// ---- FBs/Zaptec ECS/Client FBs/FB_ECS_HTTP_ZaptecAccount.TcPOU
{attribute 'hide_all_locals'}
FUNCTION_BLOCK FB_ECS_HTTP_ZaptecAccount
VAR_INPUT
	bStart					: BOOL;													//Start/Stop this Functions
	byMode					: BYTE;													//Work mode : 0 = Send current to each Charger; 1 = Send current to a Installation of chargers
	sUsername				: STRING(100);											//Username from the Zaptec Account
	sPassword				: STRING(100);											//Password from the Zaptec Account
	arrCharger				: ARRAY[1..100] OF ST_Zaptec_Input_Charger;				//Structure with Data for each Charging Station
	arrInstallation			: ARRAY[1..100] OF ST_Zaptec_Input_Installation;		//Structure with Data for each Installation of Charging Stations
END_VAR
VAR_OUTPUT
	bValidResult			: BOOL;													//Valid Result received from Server
	bBusy             		: BOOL;													//Busy Flag
    bError              	: BOOL;													//Error Flag
	hrErrorCode       		: HRESULT;												//Error Result from Http Client
	arrStateCharger			: ARRAY[1..100] OF ST_Zaptec_ECS_State;					//Output Structure with the State from each Charging Station
END_VAR
VAR
	fbHttpClient        	: FB_IotHttpClient :=(sHostName:='api.zaptec.com',		//Http Client Function
                       		  bKeepAlive:=FALSE, tConnectionTimeout:=T#10S);
	fbHttpPostToken         : FB_HTTP_Post_Zaptec_ReqToken;							//Http Post to receive the Bearer Token
 	fbHttpGetChrgState		: FB_HTTP_Get_Zaptec_ECS_State;							//Http Get to receive the State from each Charging station
	fbHttpPostCurrent		: FB_HTTP_Post_Zaptec_Current;							//Http Post to control each Chrging station or a installation of charging stations with the current setpoint
	fbTaskIndex				: GETCURTASKINDEX;										//Function to find the Task Index
	timDelay				: TON;													//Timer for Delay between the Requests
	timTimout				: TON;													//Timer for Timeout in the State machine
	timToken				: TON;													//Timer to make a Request for a new Token
	FPStart					: R_TRIG;												//Internal positive Edge
	FPErrorToken			: R_TRIG;												//Internal positive Edge
	FPErrorGetState			: R_TRIG;												//Internal positive Edge
	FPErrorPostCurrent		: R_TRIG;												//Internal positive Edge
	FPErrorClient			: R_TRIG;												//Internal positive Edge
	FPTimToken				: R_TRIG;												//Internal positive Edge
	FNStart					: F_TRIG;												//Internal negative Edge
	byNumberOfChargers		: BYTE;													//Number of charging station with insert ID in the Input Array
	byNumberOfInstallation	: BYTE;													//Number of Installations with insert ID in the Input Array
	byECSInProgress			: BYTE;													//Charging station in Progress to read out the State or write the current
	byInstInProgress		: BYTE;													//Installation of charging stations in Progress to write the current
	byLPInfo				: BYTE;													//Loop Variable to define some parts in the Code
	iState					: INT;													//Variabel for state machine
	iState_CP				: INT;													//Variabel for state machine to compare it for timeout
	udiCycleTime			: UDINT;												//Cycletime in ms
END_VAR

//Creator : Kai Ebensperger
//Company : Lynus AG
//Date : 04.11.2021
//Version : 1.0.0.0

//With this Function its possible to receive information from each charging station in a Zaptec Account in there cloudplattform
//Its also possible to control the charging station with this function by a curretn setpoint.
//We can control each Cahrging station with the current or each installation with more charging stations with a sum of current
//When the Installation mode is active, then the system of the charging station distribute the sum of current among themselves
//Attention : This Function need allways the Charging IDs. Even if the current is sent to the installation. Becasue the State Get Request for each charging station its possible only with the Charging IDs
//This Function can handle maximal 100 charging stations and 100 Installations

(*------------------------------------------------------------------------------------Limits------------------------------------------------------------------------------------------------------*)

byMode := LIMIT(0,byMode,1);

(*------------------------------------------------------------------------------------Configure HTTP Client------------------------------------------------------------------------------------------------------*)

IF NOT fbHttpClient.bConfigured THEN
    fbHttpClient.nHostPort:= 443;
	fbHttpClient.stTLS.bNoServerCertCheck := TRUE;
END_IF

(*------------------------------------------------------------------------------------Logic------------------------------------------------------------------------------------------------------*)

//Calculate the number of chargers and installations from the input array
byNumberOfChargers := 0;
	byNumberOfInstallation := 0;

FOR byLPInfo := 1 TO 100 BY 1 DO
	IF arrCharger[byLPInfo].sChargerID <> '' THEN byNumberOfChargers := byNumberOfChargers + 1; END_IF 
		IF arrInstallation[byLPInfo].sInstallationID <> '' THEN byNumberOfInstallation := byNumberOfInstallation + 1; END_IF  
END_FOR 	

//Delay between the Requests
fbTaskIndex(index=> );
	udiCycleTime := TwinCAT_SystemInfoVarList._TaskInfo[fbTaskIndex.index].CycleTime / 10000;
		timDelay(IN:= , PT:= T#1MS * udiCycleTime, Q=> , ET=> );

//Timout
IF iState_CP = iState AND iState <> 0 THEN timTimout.IN := TRUE; ELSE timTimout.IN := FALSE; END_IF
	timTimout(IN:= , PT:= T#20S, Q=> , ET=> );

//Timer for the Token
//After received the validation from the Token start this timer.
//After the Delay stop the State machine and make a request for a new Token
IF fbHttpPostToken.udiValidityToken <> 0 THEN
	timToken.PT := (T#1S * (fbHttpPostToken.udiValidityToken - 600));	//Less 10 Minutes
ELSE
	timToken.PT := T#600S;
END_IF
	timToken(IN:= , PT:= , Q=> , ET=> );	

FPTimToken(CLK:= timToken.Q, Q=> );
	
//Start	
FPStart(CLK:= bStart, Q=> );
	IF FPStart.Q AND NOT fbHttpPostToken.bBusy AND NOT fbHttpGetChrgState.bBusy AND NOT fbHttpPostCurrent.bBusy AND fbHttpClient.bConfigured THEN istate := 1; END_IF
		IF NOT bStart THEN istate := 0; END_IF	

CASE iState OF

	0://Init Step	
		fbHttpPostToken.bPostToken := FALSE;
			fbHttpGetChrgState.bSend := FALSE;
				fbHttpPostCurrent.bSend := FALSE;	
					byECSInProgress := 0;
						byInstInProgress := 0;
							timToken.IN := FALSE;
								bValidResult := FALSE;
									timdelay.IN := FALSE;
		
		FOR byLPInfo := 1 TO 100 BY 1 DO					
			arrStateCharger[byLPInfo].bIsEnabled := FALSE;	
				arrStateCharger[byLPInfo].bIsOnline := FALSE;
					arrStateCharger[byLPInfo].diOperationMode := 0;	
						arrStateCharger[byLPInfo].diWarnings := 0;
							arrStateCharger[byLPInfo].rAllocatedCurrent := 0;
								arrStateCharger[byLPInfo].rMaxCurrect := 0;
									arrStateCharger[byLPInfo].rMinCurrect := 0;
										arrStateCharger[byLPInfo].rCurrentL1 := 0;	
											arrStateCharger[byLPInfo].rCurrentL2 := 0;	
												arrStateCharger[byLPInfo].rCurrentL3 := 0;	
													arrStateCharger[byLPInfo].rPower := 0;
														arrStateCharger[byLPInfo].rEnergySession := 0;		
															arrStateCharger[byLPInfo].sChargerID := '';	
		END_FOR		
				
	1://Request for Bearer Token
		iState_CP := iState;
	
		fbHttpPostToken.bPostToken := TRUE;
			timToken.IN := FALSE;
		
		IF NOT fbHttpPostToken.bBusy THEN timdelay.IN := TRUE; END_IF 
	
		IF NOT fbHttpPostToken.bBusy AND fbHttpPostToken.bValidResult AND NOT fbHttpPostToken.bError AND timdelay.Q THEN
			istate := 2; 
				timdelay.IN := FALSE;
					byECSInProgress := 1;
						byInstInProgress := 1;
							fbHttpPostToken.bPostToken := FALSE;
								timToken.IN := TRUE;
		END_IF
		
		//Valid Result
		bValidResult := fbHttpPostToken.bValidResult;
		
		//Error, Timout or Request for a new Token
		IF FPErrorToken.Q OR timTimout.Q OR FPTimToken.Q OR FPErrorClient.Q THEN istate := 300; END_IF

	2://Request for State of Each Charging Station
		iState_CP := iState;
		
		fbHttpGetChrgState.bSend := TRUE;
			fbHttpGetChrgState.sChargerID := arrCharger[byECSInProgress].sChargerID;
		
		IF NOT fbHttpGetChrgState.bBusy THEN timdelay.IN := TRUE; END_IF 
		
		IF NOT fbHttpGetChrgState.bBusy AND fbHttpGetChrgState.bValidResult AND NOT fbHttpGetChrgState.bError AND timdelay.Q THEN
			IF byMode = 0 THEN istate := 3; END_IF
				IF byMode = 1 THEN istate := 4; END_IF
					timdelay.IN := FALSE;
						arrStateCharger[byECSInProgress] := fbHttpGetChrgState.stChargerStates;
							fbHttpGetChrgState.bSend := FALSE;	
		END_IF
		
		//Valid Result
		bValidResult := fbHttpGetChrgState.bValidResult;
		
		//Error, Timout or Request for a new Token
		IF FPErrorGetState.Q OR timTimout.Q OR FPTimToken.Q OR FPErrorClient.Q THEN istate := 300; END_IF
		
	3://Write current to charging station
		iState_CP := iState;
		
		fbHttpPostCurrent.bSend := TRUE;
			fbHttpPostCurrent.sID := arrCharger[byECSInProgress].sChargerID;
				fbHttpPostCurrent.rMaxCurrentCharger := arrCharger[byECSInProgress].rMaxCurrentCharger;
 					fbHttpPostCurrent.rMinCurrentCharger := arrCharger[byECSInProgress].rMinCurrentCharger;
		
		IF NOT fbHttpPostCurrent.bBusy THEN timdelay.IN := TRUE; END_IF 
		
		IF NOT fbHttpPostCurrent.bBusy AND fbHttpPostCurrent.bValidResult AND NOT fbHttpPostCurrent.bError AND timdelay.Q THEN
			iState := 5;
				timdelay.IN := FALSE;
					fbHttpPostCurrent.bSend := FALSE;	
		END_IF
		
		//Valid Result
		bValidResult := fbHttpPostCurrent.bValidResult;
		
		//Error, Timout or Request for a new Token
		IF FPErrorPostCurrent.Q OR timTimout.Q OR FPTimToken.Q OR FPErrorClient.Q THEN istate := 300; END_IF
		
	4://Write current to installation of charging stations	
		iState_CP := iState;	
	
		fbHttpPostCurrent.bSend := TRUE;
			fbHttpPostCurrent.sID := arrInstallation[byInstInProgress].sInstallationID;
				fbHttpPostCurrent.rAvailableCurrentInstallation := arrInstallation[byInstInProgress].rAvailableCurrentInstallation;
		
		IF NOT fbHttpPostCurrent.bBusy THEN timdelay.IN := TRUE; END_IF 
		
		IF NOT fbHttpPostCurrent.bBusy AND fbHttpPostCurrent.bValidResult AND NOT fbHttpPostCurrent.bError AND timdelay.Q THEN
			iState := 5;
				timdelay.IN := FALSE;
					fbHttpPostCurrent.bSend := FALSE;	
		END_IF
		
		//Valid Result
		bValidResult := fbHttpPostCurrent.bValidResult;
		
		//Error, Timout or Request for a new Token
		IF FPErrorPostCurrent.Q OR timTimout.Q OR FPTimToken.Q OR FPErrorClient.Q THEN istate := 300; END_IF
		
	5://Next charging station and next installation	
		iState_CP := iState;
		
		byECSInProgress := byECSInProgress + 1;
		byInstInProgress := byInstInProgress + 1;
		
		//Back to read out next state from charging station
		iState := 2;
		
		IF byECSInProgress > byNumberOfChargers THEN byECSInProgress := 1; END_IF
			IF byInstInProgress > byNumberOfInstallation THEN byInstInProgress := 1; END_IF  	
		
		//Reset Error
		bError := FALSE;
			
	300://Error or restart after receive a new Token
		iState_CP := iState;
		
		timdelay.IN := FALSE;
			fbHttpPostToken.bPostToken := FALSE;
				fbHttpGetChrgState.bSend := FALSE;
					fbHttpPostCurrent.bSend := FALSE;	
						byECSInProgress := 0;
							byInstInProgress := 0;
								bError := TRUE;
								//Restart
								IF NOT fbHttpPostToken.bBusy AND NOT fbHttpGetChrgState.bBusy AND NOT fbHttpPostCurrent.bBusy THEN 
									istate := 1;
								END_IF	
		
		
END_CASE		
		
(*------------------------------------------------------------------------------------HTTP Functions------------------------------------------------------------------------------------------------------*)

fbHttpPostToken(
	sUsername:= sUsername, 
	sPassword:= sPassword, 
	bPostToken:= , 
	tTimeOut:= T#20S,
	fbClient:= fbHttpClient, 
	bValidResult=> , 
	bBusy=> , 
	bError=> , 
	udiValidityToken=> , 
	sToken=> , 
	sTokenType=> );

FPErrorToken(CLK:= fbHttpPostToken.bError, Q=> );
	
fbHttpGetChrgState(
	bSend:= , 
	sToken:= fbHttpPostToken.sToken, 
	sTokenType:= fbHttpPostToken.sTokenType, 
	sChargerID:= , 
	tTimeOut:= T#20S,
	fbClient:= fbHttpClient, 
	bValidResult=> , 
	bBusy=> , 
	bError=> , 
	stChargerStates=> );

FPErrorGetState(CLK:= fbHttpGetChrgState.bError, Q=> );
	
fbHttpPostCurrent(
	bSend:= , 
	byMode:= byMode, 
	rMaxCurrentCharger:= , 
	rMinCurrentCharger:= , 
	rAvailableCurrentInstallation:= , 
	sToken:= fbHttpPostToken.sToken, 
	sTokenType:= fbHttpPostToken.sTokenType, 
	sID:= , 
	tTimeOut:= T#20S,
	fbClient:= fbHttpClient, 
	bValidResult=> , 
	bBusy=> , 
	bError=> );

FPErrorPostCurrent(CLK:= fbHttpPostCurrent.bError, Q=> );	

//Http Client
FNStart(CLK:= bStart, Q=> );
	IF FNStart.Q THEN fbHttpClient.Disconnect(); END_IF

fbHttpClient.Execute();

FPErrorClient(CLK:= fbHttpClient.bError, Q=> );

//Busy
IF fbHttpPostToken.bBusy OR fbHttpGetChrgState.bBusy OR fbHttpPostCurrent.bBusy THEN bBusy := TRUE; ELSE bBusy := FALSE; END_IF  

//Error
hrErrorCode := fbHttpClient.hrErrorCode;

END_FUNCTION_BLOCK

// ---- FBs/Zaptec ECS/Helper FBs/FB_HTTP_Post_Zaptec_ReqToken.TcPOU
{attribute 'hide_all_locals'}
{attribute 'conditionalshow'}
FUNCTION_BLOCK FB_HTTP_Post_Zaptec_ReqToken
VAR_INPUT
	{attribute 'hide'}
	sUsername			: STRING(100);											//Username from the Zaptec Account
	{attribute 'hide'}
	sPassword			: STRING(100);											//Password from the Zaptec Account
	{attribute 'hide'}
    bPostToken          : BOOL;													//Send Post Request for Token		
	{attribute 'hide'}
	tTimeOut			: TIME := T#10S;										//Timer for Timeout
END_VAR
VAR_IN_OUT
	{attribute 'hide'}
    fbClient            : FB_IotHttpClient;										//FB Http Client
END_VAR
VAR_OUTPUT
	{attribute 'hide'}
	bValidResult		: BOOL;													//Valid Result received from Server
	{attribute 'hide'}
	bBusy             	: BOOL;													//Busy Flag
	{attribute 'hide'}
    bError              : BOOL;													//Error Flag
	{attribute 'hide'}
	udiValidityToken	: UDINT;												//Validity from the Token in seconds. (Token is valid only for this time)
	{attribute 'hide'}
	sToken				: STRING(1500);											//Bearer Token
	{attribute 'hide'}
	sTokenType			: STRING(50);											//Token Type
END_VAR
VAR
	fbJsonRead			: FB_JsonDomParser;										//Json Parser
	jsonDoc		  		: SJsonValue;											//Json Value
	jsonProp			: SJsonValue;											//Json Value
    fbRequest           : FB_IotHttpRequest;									//HTTP Request
	fbHeader            : FB_IotHttpHeaderFieldMap;								//Header Function
	timTimeout			: TON;													//Timer for Timeout
    RisingEdge          : R_TRIG;												//Internal Risig Edge
    bOnce               : BOOL:= TRUE;											//Add the addidional Header Part
    bGetContentResult   : BOOL;													//Content Received
 	nState              : UDINT;												//State
	nReqCount           : UDINT;												//Request Counter
    nResCount           : UDINT;												//Receive Conter
    nValidResCount      : UDINT;												//Valid receive Counter
    nErrCount           : UDINT;												//Error Counter
	sUsernameInt		: STRING(200);											//Internal Username
	sPasswordInt		: STRING(200);											//Internal Password
   	sContent            : STRING(500);											//Content to send with the psot request
	sReceiveContent		: STRING(2000);											//Received Content
END_VAR

//Creator : Kai Ebensperger
//Company : Lynus AG
//Date : 03.11.2021
//Version : 1.0.0.0

//With this Function is possible to make a POST Request to a Zaptec Account to receive the Bearer Token
//This Token is neccessary for all other Requests to the Zaptec Account
//Each Token has a Validity

RisingEdge(CLK:= bPostToken);

//Content with Username and PW
sUsernameInt := sUsername;
sPasswordInt := sPassword;

//URL Encoding for Username
IF FIND(sUsernameInt,'@') <> 0 THEN
	sUsernameInt := REPLACE(sUsernameInt,'%40',1,FIND(sUsernameInt,'@'));
END_IF

//URL Encoding for Password
IF FIND(sPasswordInt,'@') <> 0 THEN
	sPasswordInt := REPLACE(sPasswordInt,'%40',1,FIND(sPasswordInt,'@'));
END_IF

//Prepear the Payload for the Post Request to receive the Token
sContent := 'grant_type=password&username=';
	CONCAT2(ADR(sContent),ADR(sUsernameInt),ADR(sContent),SIZEOF(sContent));
		sContent := CONCAT(sContent,'&password=');
			CONCAT2(ADR(sContent),ADR(sPasswordInt),ADR(sContent),SIZEOF(sContent));

//Add the Content type in the Header
IF bOnce THEN
    fbHeader.AddField('content-type','application/x-www-form-urlencoded', FALSE);
    bOnce:= FALSE;
END_IF

//Timer for Timeout
timTimeout(IN:= nState = 1 AND bBusy, PT:= tTimeOut, Q=> , ET=> );
	IF timTimeout.Q THEN nState := 0; bBusy := FALSE; END_IF

CASE nState OF
	
	0://Request
		IF RisingEdge.Q THEN
			IF fbRequest.SendRequest(sUri:= '/oauth/token', fbClient:= fbClient, 
									 eRequestType:= ETcIotHttpRequestType.HTTP_POST, 
									 pContent:= ADR(sContent), 
									 nContentSize:= LEN2(ADR(sContent)), fbHeader) THEN
				nState:= 1;
				nReqCount:= nReqCount+1;
				bBusy:= TRUE;
				bError:= FALSE;
				bValidResult := FALSE;
			END_IF
		END_IF
		
	1://Wait for the Response
		IF NOT fbRequest.bBusy THEN
			bError:= TRUE;
			IF NOT fbRequest.bError THEN
				bGetContentResult:= fbRequest.GetContent(pContent:= ADR(sReceiveContent),
														 nContentSize:= SIZEOF(sReceiveContent), 
														 bSetNullTermination:= TRUE);
				IF fbRequest.nStatusCode >= 200 AND fbRequest.nStatusCode < 300 THEN
					bValidResult := TRUE;
					//Parse Document
					jsonDoc := fbJsonRead.ParseDocument(sReceiveContent);
						//Token
						jsonProp := fbJsonRead.FindMember(jsonDoc,'access_token');
							IF jsonProp <> 0 AND fbJsonRead.IsString(jsonProp) THEN
								fbJsonRead.CopyString(jsonProp,sToken,SIZEOF(sToken));	
							END_IF
						//Token Type
						jsonProp := fbJsonRead.FindMember(jsonDoc,'token_type');
							IF jsonProp <> 0 AND fbJsonRead.IsString(jsonProp) THEN
								sTokenType := fbJsonRead.GetString(jsonProp);	
							END_IF	
						//Expires IN
						jsonProp := fbJsonRead.FindMember(jsonDoc,'expires_in');
							IF jsonProp <> 0 AND fbJsonRead.IsUint(jsonProp) THEN
								udiValidityToken := fbJsonRead.GetUint(jsonProp);	
							END_IF
					bError:= FALSE;   
					nResCount:= nResCount+1;
				END_IF
			END_IF
				nState:= 0;
				bBusy:= FALSE;
					IF bError THEN
						nErrCount:= nErrCount+1;
					END_IF
		END_IF
		
END_CASE

END_FUNCTION_BLOCK

// ---- FBs/Zaptec ECS/Helper FBs/FB_HTTP_Get_Zaptec_ECS_State.TcPOU
{attribute 'hide_all_locals'}
{attribute 'conditionalshow'}
FUNCTION_BLOCK FB_HTTP_Get_Zaptec_ECS_State
VAR_INPUT
	{attribute 'hide'}
	bSend              	 	: BOOL;													//Send the Request to the Service
	{attribute 'hide'}
	sToken					: STRING(1500);											//Bearer Token
	{attribute 'hide'}
	sTokenType				: STRING(50);											//Token Type
	{attribute 'hide'}
	sChargerID				: STRING(50);											//Charger ID
	{attribute 'hide'}
	tTimeOut				: TIME := T#10S;										//Timer for Timeout
END_VAR
VAR_IN_OUT
	{attribute 'hide'}
    fbClient            	: FB_IotHttpClient;										//Connection to the HTTP Client Function
END_VAR
VAR_OUTPUT
	{attribute 'hide'}
	bValidResult			: BOOL;													//Valid Result received from Server
	{attribute 'hide'}
	bBusy               	: BOOL;													//Function is Busy
	{attribute 'hide'}
	bError             		: BOOL;													//Function has a error
	{attribute 'hide'}
	stChargerStates			: ST_Zaptec_ECS_State;									//Structure with the States of the charging station
END_VAR
VAR
	fbJsonRead				: FB_JsonDomParser;										//Json Parser
	jsonInt		  			: SJsonValue;											//Json Value
	jsonDoc		  			: SJsonValue;											//Json Value
	jsonStateID		 		: SJsonValue;											//Json Value
	jsonIteratorArrayStart	: SJsonAIterator;										//Json AIterator
	jsonIteratorArrayEnd	: SJsonAIterator;										//Json AIterator
	fbRequest           	: FB_IotHttpRequest;									//Http Request Function
    fbHeader            	: FB_IotHttpHeaderFieldMap;								//Header Function
	timTimeout				: TON;													//Timer for Timeout
 	RisingEdge         	 	: R_TRIG;												//Internal rising edge
	diStateID				: DINT;													//State ID
   	bGetContentResult  	 	: BOOL;													//True when we receive content												
    nState             	 	: UDINT;												//Statemachine for the http request
    nReqCount          	 	: UDINT;												//Request Counter
    nResCount           	: UDINT;												//Receive Counter
    nValidResCount      	: UDINT;												//Valid Receive Counter
    nErrCount           	: UDINT;												//Error Counter
    bOnce               	: BOOL:= TRUE;											//Add the addidional Header Part
	sBearerToken			: STRING(1600);											//Bearer Token
	sBearerToken_CP			: STRING(1600);											//Bearer Token
	sContent            	: STRING(15000);										//Received Content
	sUri					: STRING;												//URL for the Request
	sValueAsString			: STRING(255);											//received Value as a String
END_VAR

//Creator : Kai Ebensperger
//Company : Lynus AG
//Date : 03.11.2021
//Version : 1.0.0.0

//With this Function its possible to make a State Request to a Charging Station in the Zaptec Account.
//To use this Function is neccessary to call first a Bearer Token for this Zaptec Account with the Post Request Function
//This Function deliver follow Information =>
//Online Stat
//Enable State
//Set Current
//Warnings
//Operation State

//Prepear Bearer Token
sTokenType := CONCAT(sTokenType,' ');
	CONCAT2(ADR(sTokenType),ADR(sToken),ADR(sBearerToken),SIZEOF(sBearerToken));

//Add the Bearer Token to the Header
IF sBearerToken <> sBearerToken_CP AND nState = 0 THEN bOnce := TRUE; sBearerToken_CP := sBearerToken; END_IF  

IF bOnce THEN
    fbHeader.AddField('Authorization',sBearerToken, FALSE);
    bOnce:= FALSE;
END_IF

//Timer for Timeout
timTimeout(IN:= nState = 1 AND bBusy, PT:= tTimeOut, Q=> , ET=> );
	IF timTimeout.Q THEN nState := 0; bBusy := FALSE; END_IF

//Statemachine to generate the Request

sUri := CONCAT(CONCAT('/api/chargers/',sChargerID),'/state');

RisingEdge(CLK:= bSend);
	CASE nState OF
		
		0://Request
			IF RisingEdge.Q THEN
				IF fbRequest.SendRequest(sUri:= sUri, fbClient:= fbClient, 
										 eRequestType:= ETcIotHttpRequestType.HTTP_GET, 0, 0, fbHeader) THEN
					nState:= 1;
					nReqCount:= nReqCount + 1;
					bBusy:= TRUE;
					bError:= FALSE;
					bValidResult := FALSE;
				END_IF
			END_IF
			
		1://Wait for the Response
			IF NOT fbRequest.bBusy THEN
				bError:= TRUE;
					IF NOT fbRequest.bError THEN
						bGetContentResult:= fbRequest.GetContent(pContent:= ADR(sContent),
																 nContentSize:= SIZEOF(sContent), 
																 bSetNullTermination:= TRUE);
						IF fbRequest.nStatusCode >= 200 AND fbRequest.nStatusCode < 300 THEN
							bValidResult := TRUE;
							nResCount:= nResCount + 1;
							bError:= FALSE;
							//Parse Document
							jsonInt := fbJsonRead.ParseDocument(sContent);
								IF jsonInt <> 0 THEN
									IF fbJsonRead.IsArray(jsonInt) THEN
										jsonIteratorArrayStart := fbJsonRead.ArrayBegin(jsonInt);	
											jsonIteratorArrayEnd := fbJsonRead.ArrayEnd(jsonInt);
									ELSE
										bError := TRUE;
									END_IF
								ELSE
									bError := TRUE;
								END_IF
									//Start to Decode the Json File
									IF jsonInt <> 0 AND jsonIteratorArrayStart <> 0 AND jsonIteratorArrayEnd <> 0 AND NOT bError THEN
										WHILE jsonIteratorArrayStart <> jsonIteratorArrayEnd DO  
											jsonDoc := fbJsonRead.GetArrayValue(jsonIteratorArrayStart);
												//Find Charger ID
												jsonStateID := fbJsonRead.FindMember(jsonDoc, 'ChargerId');
													IF jsonStateID <> 0 THEN
														IF fbJsonRead.IsString(jsonStateID) THEN	
															stChargerStates.sChargerID := fbJsonRead.GetString(jsonStateID);
														ELSE
															bError := TRUE;
														END_IF
													END_IF
												//Find State ID
												jsonStateID := fbJsonRead.FindMember(jsonDoc, 'StateId');	
													IF jsonStateID <> 0 THEN
														IF fbJsonRead.IsInt(jsonStateID) THEN
															diStateID := fbJsonRead.GetInt(jsonStateID);
																//Online State
																IF diStateID = -2 THEN 	
																	jsonStateID := fbJsonRead.FindMember(jsonDoc, 'ValueAsString');	
																		IF jsonStateID <> 0 THEN 
																			IF fbJsonRead.IsString(jsonStateID) THEN
																				IF fbJsonRead.GetString(jsonStateID) = '0' THEN
																					stChargerStates.bIsOnline := FALSE;
																				ELSIF fbJsonRead.GetString(jsonStateID) = '1' THEN 
																					stChargerStates.bIsOnline := TRUE;
																				END_IF 	
																			ELSE
																				bError := TRUE;	
																			END_IF
																		ELSE
																			bError := TRUE;
																		END_IF
																END_IF
																//Actual Current L1
																IF diStateID = 507 THEN 	
																	jsonStateID := fbJsonRead.FindMember(jsonDoc, 'ValueAsString');	
																		IF jsonStateID <> 0 THEN  
																			IF fbJsonRead.IsString(jsonStateID) THEN
																				sValueAsString := fbJsonRead.GetString(jsonStateID);
																					stChargerStates.rCurrentL1 := STRING_TO_REAL(sValueAsString);
																			ELSE
																				bError := TRUE;	
																			END_IF
																		ELSE
																			bError := TRUE;
																		END_IF
																END_IF
																//Actual Current L2
																IF diStateID = 508 THEN 	
																	jsonStateID := fbJsonRead.FindMember(jsonDoc, 'ValueAsString');
																		IF jsonStateID <> 0 THEN 	
																			IF fbJsonRead.IsString(jsonStateID) THEN
																				sValueAsString := fbJsonRead.GetString(jsonStateID);
																					stChargerStates.rCurrentL2 := STRING_TO_REAL(sValueAsString);
																			ELSE
																				bError := TRUE;	
																			END_IF
																		ELSE
																			bError := TRUE;
																		END_IF
																END_IF
																//Actual Current L3
																IF diStateID = 509 THEN 	
																	jsonStateID := fbJsonRead.FindMember(jsonDoc, 'ValueAsString');	
																		IF jsonStateID <> 0 THEN 
																			IF fbJsonRead.IsString(jsonStateID) THEN
																				sValueAsString := fbJsonRead.GetString(jsonStateID);
																					stChargerStates.rCurrentL3 := STRING_TO_REAL(sValueAsString);
																			ELSE
																				bError := TRUE;	
																			END_IF
																		ELSE
																			bError := TRUE;
																		END_IF
																END_IF
																//Max Current
																IF diStateID = 510 THEN 	
																	jsonStateID := fbJsonRead.FindMember(jsonDoc, 'ValueAsString');	
																		IF jsonStateID <> 0 THEN 
																			IF fbJsonRead.IsString(jsonStateID) THEN
																				sValueAsString := fbJsonRead.GetString(jsonStateID);
																					stChargerStates.rMaxCurrect := STRING_TO_REAL(sValueAsString);
																			ELSE
																				bError := TRUE;	
																			END_IF
																		ELSE
																			bError := TRUE;
																		END_IF
																END_IF
																//Min Current
																IF diStateID = 511 THEN 	
																	jsonStateID := fbJsonRead.FindMember(jsonDoc, 'ValueAsString');	
																		IF jsonStateID <> 0 THEN 
																			IF fbJsonRead.IsString(jsonStateID) THEN
																				sValueAsString := fbJsonRead.GetString(jsonStateID);
																					stChargerStates.rMinCurrect := STRING_TO_REAL(sValueAsString);
																			ELSE
																				bError := TRUE;	
																			END_IF
																		ELSE
																			bError := TRUE;
																		END_IF
																END_IF
																//Actual Power
																IF diStateID = 513 THEN 	
																	jsonStateID := fbJsonRead.FindMember(jsonDoc, 'ValueAsString');	
																		IF jsonStateID <> 0 THEN 
																			IF fbJsonRead.IsString(jsonStateID) THEN
																				sValueAsString := fbJsonRead.GetString(jsonStateID);
																					stChargerStates.rPower := STRING_TO_REAL(sValueAsString);
																						stChargerStates.rPower := stChargerStates.rPower / 1000;	
																			ELSE
																				bError := TRUE;	
																			END_IF
																		ELSE
																			bError := TRUE;
																		END_IF
																END_IF
																//Energy from actual/last session
																//This not allwas has the member ValueAsString, so on this point no error
																IF diStateID = 553 THEN 	
																	jsonStateID := fbJsonRead.FindMember(jsonDoc, 'ValueAsString');
																		IF jsonStateID <> 0 THEN
																			IF fbJsonRead.IsString(jsonStateID) THEN
																				sValueAsString := fbJsonRead.GetString(jsonStateID);
																					stChargerStates.rEnergySession := STRING_TO_REAL(sValueAsString);
																			ELSE
																				bError := TRUE;	
																			END_IF
																		END_IF
																END_IF
																//Allocated Currect
																IF diStateID = 708 THEN 	
																	jsonStateID := fbJsonRead.FindMember(jsonDoc, 'ValueAsString');	
																		IF jsonStateID <> 0 THEN 
																			IF fbJsonRead.IsString(jsonStateID) THEN
																				sValueAsString := fbJsonRead.GetString(jsonStateID);
																					stChargerStates.rAllocatedCurrent := STRING_TO_REAL(sValueAsString);
																			ELSE
																				bError := TRUE;	
																			END_IF
																		ELSE
																			bError := TRUE;
																		END_IF
																END_IF
																//Operation State
																IF diStateID = 710 THEN 	
																	jsonStateID := fbJsonRead.FindMember(jsonDoc, 'ValueAsString');	
																		IF jsonStateID <> 0 THEN 
																			IF fbJsonRead.IsString(jsonStateID) THEN
																				sValueAsString := fbJsonRead.GetString(jsonStateID);
																					stChargerStates.diOperationMode := STRING_TO_DINT(sValueAsString);
																			ELSE
																				bError := TRUE;	
																			END_IF
																		ELSE
																			bError := TRUE;
																		END_IF
																END_IF
																//Enabled State
																IF diStateID = 711 THEN 	
																	jsonStateID := fbJsonRead.FindMember(jsonDoc, 'ValueAsString');	
																		IF jsonStateID <> 0 THEN 
																			IF fbJsonRead.IsString(jsonStateID) THEN
																				IF fbJsonRead.GetString(jsonStateID) = '0' THEN
																					stChargerStates.bIsEnabled := FALSE;
																				ELSIF fbJsonRead.GetString(jsonStateID) = '1' THEN 
																					stChargerStates.bIsEnabled := TRUE;
																				END_IF 	
																			ELSE
																				bError := TRUE;	
																			END_IF
																		ELSE
																			bError := TRUE;
																		END_IF
																END_IF
																//Warnings
																IF diStateID = 804 THEN 	
																	jsonStateID := fbJsonRead.FindMember(jsonDoc, 'ValueAsString');	
																		IF jsonStateID <> 0 THEN 
																			IF fbJsonRead.IsString(jsonStateID) THEN
																				sValueAsString := fbJsonRead.GetString(jsonStateID);
																					stChargerStates.diWarnings := STRING_TO_DINT(sValueAsString);
																			ELSE
																				bError := TRUE;	
																			END_IF
																		ELSE
																			bError := TRUE;
																		END_IF
																END_IF
														ELSE
															bError := TRUE;	
														END_IF	
													END_IF 		
														//Next Part from Array
														jsonIteratorArrayStart := fbJsonRead.NextArray(jsonIteratorArrayStart);
										END_WHILE		
									END_IF
						END_IF
					END_IF
						nState:= 0;
						bBusy:= FALSE;
							IF bError THEN
								nErrCount:= nErrCount + 1;
							END_IF
			END_IF
			
	END_CASE

END_FUNCTION_BLOCK

// ---- FBs/Zaptec ECS/Helper FBs/FB_HTTP_Post_Zaptec_Current.TcPOU
{attribute 'hide_all_locals'}
{attribute 'conditionalshow'}
FUNCTION_BLOCK FB_HTTP_Post_Zaptec_Current
VAR_INPUT
	{attribute 'hide'}
	bSend              					: BOOL;													//Send the Request to the Service
	{attribute 'hide'}
	byMode								: BYTE;													//Work mode : 0 = Send to Charger; 1 = Send to Installation
	{attribute 'hide'}
	rMaxCurrentCharger					: REAL;													//Max Current for Charging Station 
	{attribute 'hide'}
	rMinCurrentCharger					: REAL;													//Min Current for Charging Station
	{attribute 'hide'}
	rAvailableCurrentInstallation		: REAL;													//Available Current for Installation
	{attribute 'hide'}
	sToken								: STRING(1500);											//Bearer Token
	{attribute 'hide'}
	sTokenType							: STRING(50);											//Token Type
	{attribute 'hide'}
	sID									: STRING(50);											//Charger ID or Installation ID		
	{attribute 'hide'}
	tTimeOut							: TIME := T#10S;										//Timer for Timeout
END_VAR
VAR_IN_OUT
	{attribute 'hide'}
    fbClient            				: FB_IotHttpClient;										//FB Http Client
END_VAR
VAR_OUTPUT
	{attribute 'hide'}
	bValidResult						: BOOL;													//Valid Result received from Server
	{attribute 'hide'}
	bBusy             					: BOOL;													//Busy Flag
	{attribute 'hide'}
    bError              				: BOOL;													//Error Flag
END_VAR
VAR
	fbJsonWrite     					: FB_JsonSaxWriter;	
    fbRequest           				: FB_IotHttpRequest;									//HTTP Request
	fbHeader            				: FB_IotHttpHeaderFieldMap;								//Header Function
	timTimeout							: TON;													//Timer for Timeout
    RisingEdge          				: R_TRIG;												//Internal Risig Edge
    bOnce               				: BOOL:= TRUE;											//Add the addidional Header Part
    bGetContentResult   				: BOOL;													//Content Received
 	nState              				: UDINT;												//State
	nReqCount           				: UDINT;												//Request Counter
    nResCount           				: UDINT;												//Receive Conter
    nValidResCount      				: UDINT;												//Valid receive Counter
    nErrCount           				: UDINT;												//Error Counter
	sBearerToken						: STRING(1600);											//Bearer Token
	sBearerToken_CP						: STRING(1600);											//Bearer Token
   	sContent            				: STRING(500);											//Content to send with the psot request
	sReceiveContent						: STRING(1000);											//Received Content
	sUri								: STRING;												//URL for the Request
END_VAR

//Creator : Kai Ebensperger
//Company : Lynus AG
//Date : 03.11.2021
//Version : 1.0.0.0

//With this Function is possible to make a POST Request to a Zaptec Account to set the max current on each Charging station or the complete Charge current for a installation
//With the Input byMode its possible to switch between the 2 modes
//When we send the current to a installation, then the Zaptec charging station logic distributes this electricity to the charging stations in the installation.
//In a Installation can be more then 1 Charging stations
//When we use byMode = 0 then at the sID we need the Chargig station ID
//When we use byMode = 1 then at the sID we need the Installation ID

//Limits
byMode := LIMIT(0,byMode,1);
	rMaxCurrentCharger := LIMIT(0,rMaxCurrentCharger,32);
		rMinCurrentCharger := LIMIT(6,rMinCurrentCharger,10);
			rAvailableCurrentInstallation := LIMIT(0,rAvailableCurrentInstallation,1000);	

RisingEdge(CLK:= bSend);

//Prepear Bearer Token
sTokenType := CONCAT(sTokenType,' ');
	CONCAT2(ADR(sTokenType),ADR(sToken),ADR(sBearerToken),SIZEOF(sBearerToken));

//Add the Bearer Token to the Header
IF sBearerToken <> sBearerToken_CP AND nState = 0 THEN bOnce := TRUE; sBearerToken_CP := sBearerToken; END_IF  

IF bOnce THEN
    fbHeader.AddField('Authorization',sBearerToken, FALSE);
	fbHeader.AddField('Content-type','application/json-patch+json', FALSE);
    bOnce:= FALSE;
END_IF

//Prepear URI
IF byMode = 0 THEN 
	sUri := CONCAT(CONCAT('/api/chargers/',sID),'/update');
ELSIF byMode = 1 THEN
	sUri := CONCAT(CONCAT('/api/installation/',sID),'/update');	
END_IF

//Prepear Content
IF byMode = 0 THEN 
	fbJsonWrite.StartObject();
	fbJsonWrite.AddKey('maxChargeCurrent');
	fbJsonWrite.AddReal(rMaxCurrentCharger);
	fbJsonWrite.AddKey('minChargeCurrent');
	fbJsonWrite.AddReal(rMinCurrentCharger);
	fbJsonWrite.EndObject();
	sContent := fbJsonWrite.GetDocument();
	fbJsonWrite.ResetDocument();
ELSIF byMode = 1 THEN
	fbJsonWrite.StartObject();
	fbJsonWrite.AddKey('availableCurrent');
	fbJsonWrite.AddReal(rAvailableCurrentInstallation);
	fbJsonWrite.EndObject();
	sContent := fbJsonWrite.GetDocument();
	fbJsonWrite.ResetDocument();
END_IF

//Timer for Timeout
timTimeout(IN:= nState = 1 AND bBusy, PT:= tTimeOut, Q=> , ET=> );
	IF timTimeout.Q THEN nState := 0; bBusy := FALSE; END_IF

CASE nState OF
	
	0://Request
		IF RisingEdge.Q THEN
			IF fbRequest.SendRequest(sUri:= sUri, fbClient:= fbClient, 
									 eRequestType:= ETcIotHttpRequestType.HTTP_POST, 
									 pContent:= ADR(sContent), 
									 nContentSize:= LEN2(ADR(sContent)), fbHeader) THEN
				nState:= 1;
				nReqCount:= nReqCount+1;
				bBusy:= TRUE;
				bError:= FALSE;
				bValidResult := FALSE;
			END_IF
		END_IF
		
	1://Wait for the Response
		IF NOT fbRequest.bBusy THEN
			bError:= TRUE;
			IF NOT fbRequest.bError THEN
				bGetContentResult:= fbRequest.GetContent(pContent:= ADR(sReceiveContent),
														 nContentSize:= SIZEOF(sReceiveContent), 
														 bSetNullTermination:= TRUE);
				IF fbRequest.nStatusCode >= 200 AND fbRequest.nStatusCode < 300 THEN
					bValidResult := TRUE;
					bError:= FALSE;   
					nResCount:= nResCount+1;
				END_IF
			END_IF
				nState:= 0;
				bBusy:= FALSE;
					IF bError THEN
						nErrCount:= nErrCount+1;
					END_IF
		END_IF
		
END_CASE

END_FUNCTION_BLOCK
